Universal Robots PolyScope program: GrabNozzleAndStandby.urp

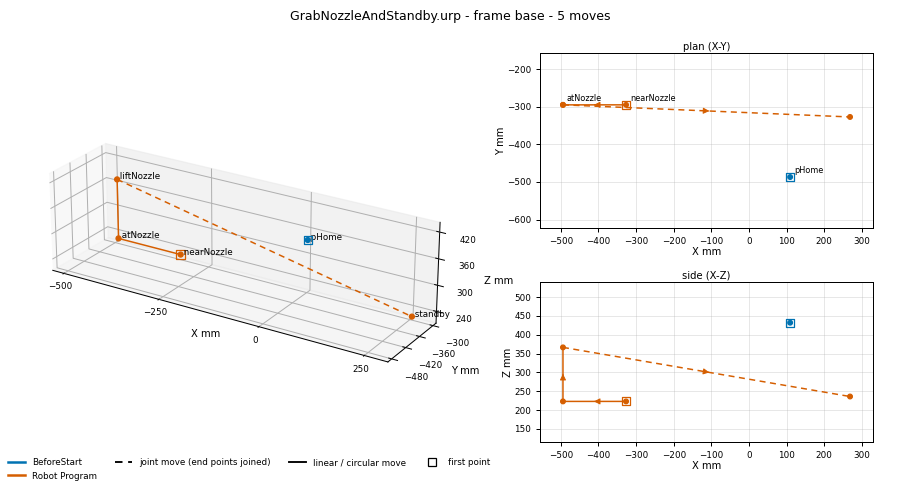
[picture p0: tool path of GrabNozzleAndStandby.urp in frame base, 5 of 5 moves have a stored position in this frame; points joined in program order, loops and branches not executed]
Program GrabNozzleAndStandby (installation=admin directory=/programs/TestProgram/PickAndPlaceTesting createdIn=3.15.8.106339 lastSavedIn=3.15.8.106339 robotSerialNumber=2015350926)
Calibrated DH parameters: a=[0, -0.425, -0.39225, 0, 0, 0]; d=[0.089159, 0, 0, 0.10915, 0.09465, 0.0823]; alpha=[1.570796, 0, 0, 1.570796, -1.570796, 0]; deltaTheta=[0, 0, 0, 0, 0, 0]
BeforeStart
  MoveJ speed 60 deg/s, acceleration 80 deg/s^2 (useActiveTCP=true)
    Waypoint pHome: TCP in base x=109.152 y=-486.9 z=431.859 mm, rx=0 ry=3.1416 rz=0 rad; joints [90, -90, 90, -90, -89.998, 0] deg
Robot Program (runOnlyOnce=true)
  MoveJ speed 60 deg/s, acceleration 80 deg/s^2 (useActiveTCP=true)
    Waypoint nearNozzle: motionParameters(blendRadius=0.08); TCP in base x=-326.725 y=-295.107 z=222.846 mm, rx=-0.0001 ry=-3.1415 rz=0 rad; joints [27.735, -90.007, 122.207, -122.207, -90.001, -62.263] deg
  MoveL speed 200 mm/s, acceleration 100 mm/s^2 (useActiveTCP=true) feature=Base
    Waypoint atNozzle: TCP in base x=-494.308 y=-295.135 z=222.83 mm, rx=-0.0001 ry=3.1415 rz=-0.0001 rad; joints [19.91, -72.584, 101.479, -118.893, -89.995, -70.092] deg
    Wait Sleep waitTime=0.4
    Set DigitalOutput pin=digital_out[0]; digitalValue=1
    Wait Sleep waitTime=0.4
    Waypoint liftNozzle: motionParameters(blendRadius=0.08); TCP in base x=-494.292 y=-295.1 z=366.384 mm, rx=-0.0001 ry=3.1415 rz=-0.0001 rad; joints [19.908, -78.798, 87.208, -98.405, -89.996, -70.096] deg
  MoveJ speed 60 deg/s, acceleration 80 deg/s^2 (useActiveTCP=true)
    Waypoint standby: TCP in base x=268.306 y=-327.29 z=235.849 mm, rx=-0.0001 ry=-3.1415 rz=0 rad; joints [114.399, -93.504, 123.351, -119.846, -90.003, 24.403] deg
